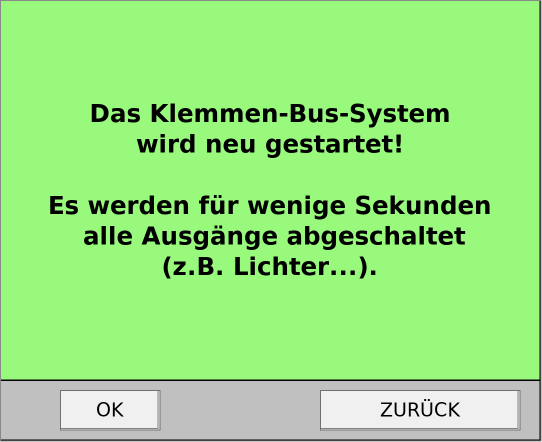
VISUALIZATION V_ECReset  // 542x442
    Rectangle (0,380 540x60)
    Button (60,390 100x40), "OK"
        OnMouseDown: toggle gfbSystemCX.VbDeviceReset
        OnMouseUp: change screen: Previous 
    Button (320,390 200x40), "ZURÜCK"
        OnMouseUp: change screen: Previous 
    Rectangle (0,0 540x380), "Das Klemmen-Bus-System wird neu gestartet! Es werden für wenige Sekunden alle Ausgänge abgeschaltet (z.B. Lichter...)."
END_VISUALIZATION

(* stored: Version 1.1.0.1, ProductVersion 3.1.4018.10
   Visu V_ECReset: Id {42dd9347-a23e-4423-91d6-7f7c7f202a6b} *)
